// TwinCAT 3 PLC project PLC
// ProgramVersion: 3.1.0.8
// libraries:
//   Tc2_Standard, * (Beckhoff Automation GmbH)
//   Tc2_System, * (Beckhoff Automation GmbH)
//   Tc3_Interfaces, * (Beckhoff Automation GmbH)
//   Tc3_Module, * (Beckhoff Automation GmbH)
// project tree:
//   GVLs/ GVL_Main.TcGVL, GVL_Offload.TcGVL, GVL_Soldering.TcGVL
//   Helper/ FB_Clock.TcPOU, FB_LiveBit.TcPOU
//   / PlcTask.TcTTO
//   POUs/ EN_SolderingSequence.TcDUT, FB_OffLoad.TcPOU, FB_Offload2.TcPOU, FB_Soldering.TcPOU, MAIN.TcPOU
//   Sequence/ EN_SequenceMode.TcDUT, EN_SequenceStartNames.TcDUT, EN_SequenceState.TcDUT, FB_Sequence.TcPOU
// real-time tasks:
//   TASK PlcTask: cycle T#10ms, priority 20, ADS port 350

CONFIGURATION PLC
    RESOURCE PLC ON TwinCAT3
        TASK PlcTask(INTERVAL := T#10ms, PRIORITY := 20);
        PROGRAM MAIN WITH PlcTask : MAIN;
    END_RESOURCE
END_CONFIGURATION

// ---- POUs/EN_SolderingSequence.TcDUT
TYPE EN_SolderingSequence :
(
	SolderingSequenceStep11 := 11,
	SolderingSequenceStep12,
	SolderingSequenceStep13,
	SolderingSequenceStep14,
	SolderingSequenceStep15,
	SolderingSequenceStep16,
	SolderingSequenceStep17,
	SolderingSequenceStep18,
	SolderingSequenceStep19,
	SolderingSequenceStep20
);
END_TYPE

// ---- Sequence/EN_SequenceMode.TcDUT
TYPE EN_SequenceMode :
(
	SequenceModeNormal := 0,
	SequenceModeStep,
	SequenceModeBreak
);
END_TYPE

// ---- Sequence/EN_SequenceStartNames.TcDUT
TYPE EN_SequenceStartNames :
(
	SequenceStartNamesStart:=10,
	SequenceStartNamesWait:=100,
	SequenceStartNamesDone:=200,
	SequenceStartNamesInit:=300,
	SequenceStartNamesStop:=400
);
END_TYPE

// ---- Sequence/EN_SequenceState.TcDUT
TYPE EN_SequenceState :
(
	SequenceStateActive := 0,
	SequenceStateError,
	SequenceStateWaiting,
	SequenceStateHalt,
	SequenceStateStop,
	SequenceStateInit,
	SequenceStateDone,
	SequenceStateStep
);
END_TYPE

// ---- GVLs/GVL_Main.TcGVL
VAR_GLOBAL
	FirstCycle				:BOOL:=TRUE;
	Clock_1_Hz				:FB_Clock;
	LiveBit					:FB_LiveBit;
END_VAR

// ---- GVLs/GVL_Offload.TcGVL
VAR_GLOBAL
	OffloadStart:BOOL;
END_VAR

// ---- GVLs/GVL_Soldering.TcGVL
VAR_GLOBAL
	SolderingStart			:BOOL;
	SolderingStop			:BOOL;
	SolderingCont			:BOOL;
	SolderingMode			:EN_SequenceMode:=SequenceModeNormal;
END_VAR

// ---- POUs/MAIN.TcPOU
PROGRAM MAIN
VAR
	i 							:INT;
	m_Fbi_Soldering				:FB_Soldering;
	m_Fbi_OffLoad				:FB_OffLoad;
	m_Fbi_OffLoad2				:FB_OffLoad2;
	m_Clock:BOOL;
	
	
END_VAR

m_Fbi_Soldering.InInit			:=FirstCycle;
m_Fbi_OffLoad.InInit			:=SolderingStart OR FirstCycle;
m_Fbi_OffLoad2.InInit			:=SolderingStart OR FirstCycle;

Clock_1_Hz.InInit				:=FirstCycle OR LiveBit.OutReTrigger;

Clock_1_Hz();

LiveBit			(	InTrigger	:=Clock_1_Hz.OutClock);

m_fbi_Soldering	(	InStart		:=SolderingStart,
					Instop		:=SolderingStop,
					InCont		:=SolderingCont,
					InMode		:=SolderingMode);
m_Fbi_OffLoad	(	InStart		:=m_fbi_Soldering.OutSequenceDone);
m_Fbi_OffLoad2	(	InStart		:=m_Fbi_OffLoad.OutSequenceDone);



FirstCycle						:=FALSE;
SolderingStart					:=FALSE;
SolderingStop					:=FALSE;
SolderingCont					:=FALSE;

END_PROGRAM

// ---- POUs/FB_Soldering.TcPOU
FUNCTION_BLOCK PUBLIC FB_Soldering EXTENDS FB_Sequence
VAR_INPUT
END_VAR
VAR_OUTPUT
END_VAR
VAR
END_VAR

SUPER^.Main();
CASE m_SequenceNumber OF
	SequenceStartNamesStart:
		StartDelaySetTime(T#5S);
		IF m_Delay.Q THEN
			SetSequenceIgnoreStop(SolderingSequenceStep11);
		END_IF
		
	SolderingSequenceStep11:
		StartDelaySetTime(T#5S);
		IF m_Delay.Q THEN
			SetSequenceIgnoreStop(SolderingSequenceStep12);
		END_IF

	SolderingSequenceStep12:
		StartDelaySetTime(T#1S);
		IF m_Delay.Q THEN
			SetSequence(SolderingSequenceStep13);
		END_IF

	SolderingSequenceStep13:
		StartDelaySetTime(T#1S);
		IF m_Delay.Q THEN
			SetSequence(SolderingSequenceStep14);
		END_IF

	SolderingSequenceStep14:
		StartDelaySetTime(T#1S);
		IF m_Delay.Q THEN
			Done();
		END_IF
	
END_CASE

END_FUNCTION_BLOCK

// ---- Sequence/FB_Sequence.TcPOU
FUNCTION_BLOCK FB_Sequence
VAR_IN_OUT
END_VAR
VAR_INPUT
	InInit						:BOOL;
	InStart						:BOOL;
	InStop						:BOOL;
	InCont						:BOOL;
	InMode						:EN_SequenceMode;
END_VAR
VAR_OUTPUT
	OutSequenceActive			:BOOL;
	OutSequenceWaiting			:BOOL;
	OutSequenceInit				:BOOL;
	OutSequenceDone				:BOOL;
	OutSequenceStop				:BOOL;

	OutSequenceState			:EN_SequenceState;
END_VAR
VAR
	m_FlStart					:BOOL;
	m_FlStop					:BOOL;
	m_FlCont					:BOOL;

	m_Delay						:TON;
	m_DelayTime					:TIME;
	m_DelayStart				:BOOL;

	m_SequenceNumber			:INT;
	m_SequenceNumberOld			:INT;
	m_SequenceLast				:INT;
	
	m_IgnoreStopActive			:BOOL;
	m_StepActive				:BOOL;

	m_SequenceState				:INT;
END_VAR

METHOD PUBLIC StartDelay : BOOL
m_DelayStart:=TRUE;
END_METHOD

METHOD PUBLIC Init : BOOL
IF InInit THEN
	m_SequenceNumber		:=SequenceStartNamesInit;
	m_SequenceLast			:=m_SequenceNumber;
	m_SequenceNumberOld		:=m_SequenceNumber;
	
	m_FlStart				:=FALSE;
	m_FlCont				:=FALSE;
	m_FlStop				:=FALSE;
	
	m_DelayStart			:=FALSE;
	m_SequenceState			:=SequenceStateInit;

END_IF
END_METHOD

METHOD PROTECTED Main : BOOL
Init();
Start();
Stop();
Cont();

IF m_SequenceNumberOld<>m_SequenceNumber THEN
	m_SequenceNumberOld		:=m_SequenceNumber;
	m_DelayStart			:=FALSE;
	m_StepActive			:=TRUE;
END_IF
m_Delay.PT					:=m_DelayTime;
m_Delay.IN					:=m_DelayStart;
m_Delay();


IF 		m_SequenceState=SequenceStateWaiting THEN
	OutSequenceActive		:=FALSE;
	OutSequenceInit			:=FALSE;
	OutSequenceWaiting		:=TRUE;
	OutSequenceDone			:=TRUE;
	OutSequenceStop			:=FALSE;
	
ELSIF 	m_SequenceState=SequenceStateInit THEN
	OutSequenceActive		:=FALSE;
	OutSequenceInit			:=TRUE;
	OutSequenceWaiting		:=FALSE;
	OutSequenceDone			:=FALSE;
	OutSequenceStop			:=FALSE;
	
ELSIF 	m_SequenceState=SequenceStateActive THEN
	OutSequenceActive		:=TRUE;
	OutSequenceInit			:=FALSE;
	OutSequenceWaiting		:=FALSE;
	OutSequenceDone			:=FALSE;
	OutSequenceStop			:=FALSE;

ELSIF 	m_SequenceState=SequenceStateStop THEN
	OutSequenceActive		:=TRUE;
	OutSequenceInit			:=FALSE;
	OutSequenceWaiting		:=FALSE;
	OutSequenceDone			:=FALSE;
	IF m_IgnoreStopActive THEN
		OutSequenceStop			:=Clock_1_Hz.OutClock;
	ELSE
		OutSequenceStop			:=TRUE;
	END_IF

ELSIF 	m_SequenceState=SequenceStateDone THEN
	OutSequenceDone			:=TRUE;
	m_SequenceState			:=SequenceStateWaiting;
	SetSequence(SequenceStartNamesWait);

END_IF

OutSequenceState			:=m_SequenceState;
END_METHOD

METHOD PUBLIC Cont : BOOL
IF InCont AND NOT m_FlCont AND m_SequenceState=SequenceStateStop THEN
	m_FlCont				:=TRUE;
	m_SequenceState			:=SequenceStateActive;
END_IF

IF NOT Incont AND m_FlCont THEN
	m_FlCont				:=FALSE;
END_IF
END_METHOD

METHOD PUBLIC SetSequenceIgnoreStop : BOOL
VAR_INPUT
	InSequence:INT;
END_VAR
IF InMode=SequenceModeNormal OR (InMode=SequenceModeStep AND InCont)  THEN
	m_SequenceLast			:=m_SequenceNumber;
	m_SequenceNumber		:=InSequence;
	m_IgnoreStopActive		:=TRUE;
END_IF

IF InMode=SequenceModeStep THEN
	m_StepActive:=FALSE;
END_IF
END_METHOD

METHOD PUBLIC IncSequence : BOOL
IF m_SequenceState<>SequenceStateStop AND InMode=SequenceModeNormal THEN
	m_SequenceLast:=m_SequenceNumber;
	m_SequenceNumber:=m_SequenceNumber + 1;
	m_StepActive			:=FALSE;
END_IF
m_IgnoreStopActive:=FALSE;
END_METHOD

METHOD PUBLIC Stop : BOOL
IF InStop AND NOT m_FlStop AND m_SequenceState=SequenceStateActive THEN
	m_FlStop				:=TRUE;
	m_SequenceState			:=SequenceStateStop;
END_IF

IF NOT InStop AND m_FlStop THEN
	m_FlStop				:=FALSE;
END_IF
END_METHOD

METHOD PUBLIC SetSequence : BOOL
VAR_INPUT
	InSequence:INT;
END_VAR
IF 	(m_SequenceState<>SequenceStateStop AND InMode=SequenceModeNormal) OR 
	(InCont AND InMode=SequenceModeStep) OR 
	(InSequence=SequenceStartNamesWait)THEN
	m_SequenceLast		:=m_SequenceNumber;
	m_SequenceNumber	:=InSequence;
END_IF
IF InMode=SequenceModeStep THEN
	m_StepActive			:=FALSE;
END_IF
m_IgnoreStopActive		:=FALSE;
END_METHOD

METHOD PRIVATE Start : BOOL
IF InStart AND NOT m_FlStart AND m_SequenceState<>SequenceStateActive THEN
	m_FlStart				:=TRUE;
	m_SequenceNumber		:=SequenceStartNamesStart;
	m_DelayStart			:=FALSE;
	m_SequenceState			:=SequenceStateActive;
END_IF
IF NOT InStart AND m_FlStart THEN
	m_FlStart				:=FALSE;
END_IF
END_METHOD

METHOD PUBLIC Done : BOOL
m_SequenceState	:=SequenceStateDone;
m_StepActive	:=FALSE;
END_METHOD

METHOD PUBLIC StartDelaySetTime : BOOL
VAR_INPUT
	Delay:TIME;
END_VAR
m_DelayTime:=Delay;
StartDelay();
END_METHOD

END_FUNCTION_BLOCK

// ---- POUs/FB_OffLoad.TcPOU
FUNCTION_BLOCK FB_OffLoad EXTENDS FB_Sequence
VAR_INPUT
END_VAR
VAR_OUTPUT
END_VAR
VAR
END_VAR

SUPER^.Main();

CASE m_SequenceNumber OF
	SequenceStartNamesStart:
		StartDelaySetTime(T#1S);
		IF m_Delay.Q THEN
			SetSequence(SolderingSequenceStep11);
		END_IF
		
	SolderingSequenceStep11:
		StartDelaySetTime(T#1S);
		IF m_Delay.Q THEN
			SetSequence(SolderingSequenceStep12);
		END_IF
	SolderingSequenceStep12:
		StartDelaySetTime(T#1S);
		IF m_Delay.Q THEN
			Done();
		END_IF
	
END_CASE

END_FUNCTION_BLOCK

// ---- POUs/FB_Offload2.TcPOU
FUNCTION_BLOCK PUBLIC FB_Offload2 EXTENDS FB_Sequence
VAR_INPUT
END_VAR
VAR_OUTPUT
END_VAR
VAR
END_VAR

SUPER^.Main();

CASE m_SequenceNumber OF
	SequenceStartNamesStart:
		StartDelaySetTime(T#1S);
		IF m_Delay.Q THEN
			SetSequence(SolderingSequenceStep11);
		END_IF
		
	SolderingSequenceStep11:
		StartDelaySetTime(T#1S);
		IF m_Delay.Q THEN
			SetSequence(SolderingSequenceStep12);
		END_IF
	SolderingSequenceStep12:
		StartDelaySetTime(T#1S);
		IF m_Delay.Q THEN
			Done();
		END_IF
	
END_CASE

END_FUNCTION_BLOCK

// ---- Helper/FB_Clock.TcPOU
FUNCTION_BLOCK PUBLIC FB_Clock
VAR_INPUT
	InInit:BOOL;
	InStart:BOOL;
	InStop:BOOL;
END_VAR
VAR_OUTPUT
	OutClock:BOOL;
END_VAR
VAR
	ImpulsHigh:TP;
	ImpulsLow:TP;
	m_Start:BOOL;
	m_Stop:BOOL;
	FlNeg1:F_TRIG;
	FlNeg2:F_TRIG;
	FlPos:R_TRIG;
	
END_VAR

FlPos		(CLK:=InInit OR InStart OR FlNeg2.Q);

ImpulsHigh	(IN:=FlPos.Q,PT:=T#1S);

FlNeg1		(CLK:=ImpulsHigh.Q);

ImpulsLow	(IN:=FlNeg1.Q,PT:=T#1S);

FlNeg2		(CLK:=ImpulsLow.Q);

OutClock:=ImpulsHigh.Q;

END_FUNCTION_BLOCK

// ---- Helper/FB_LiveBit.TcPOU
FUNCTION_BLOCK PUBLIC FB_LiveBit
VAR_INPUT
	InTrigger:BOOL;
END_VAR
VAR_OUTPUT
	OutReTrigger:BOOL;
END_VAR
VAR
	m_Tof			:TOF;
	m_PosFlk		:R_TRIG;
	m_NegFlk		:F_TRIG;
	m_Toogle		:BOOL;
	
	m_Counter:INT;
END_VAR

m_PosFlk(CLK:=InTrigger);
m_NegFlk(CLK:=InTrigger);

m_Tof(IN:=m_PosFlk.Q OR m_NegFlk.Q,PT:=T#2S);
IF NOT m_Tof.Q THEN
	m_Toogle:=NOT m_Toogle;
ELSE
	m_Toogle:=FALSE;
END_IF

END_FUNCTION_BLOCK
